Universal Robots PolyScope program: vg_palatz_cards.urp

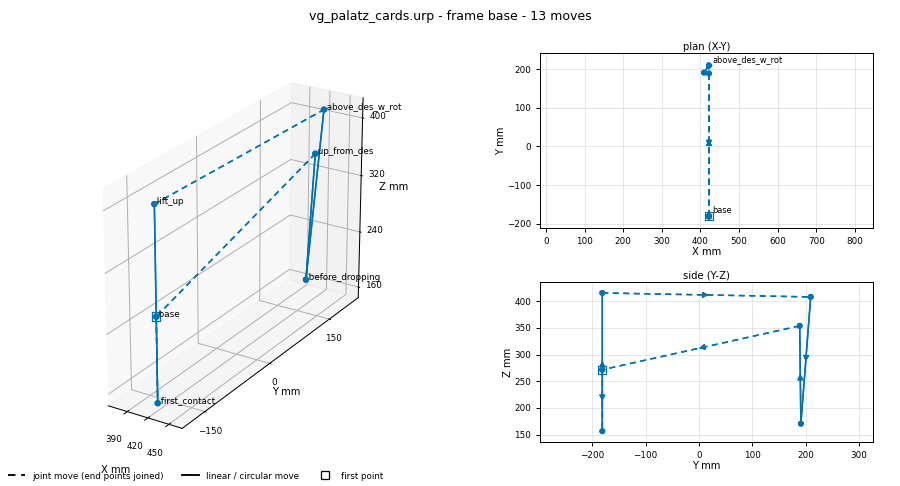
[picture p0: tool path of vg_palatz_cards.urp in frame base, 13 of 13 moves have a stored position in this frame; points joined in program order, loops and branches not executed]
Program vg_palatz_cards (installation=default directory=/programs/v_gripper_tm1326 createdIn=5.11.9.1010452 lastSavedIn=5.11.9.1010452 robotSerialNumber=20225200364)
Calibrated DH parameters: a=[0.00002, -0.569483, -0.54992, -0.00001, -0.000036, 0]; d=[0.180894, -146.691669, 192.918669, -46.053088, 0.119778, 0.115602]; alpha=[1.571425, -0.001534, 0.003359, 1.568739, -1.571477, 0]; deltaTheta=[0, 0.376258, -0.101074, -0.275185, -0.000002, 0]
Robot Program (runOnlyOnce=false)
  MoveJ speed 60 deg/s, acceleration 80 deg/s^2 (useActiveTCP=true) feature=Base
    Waypoint base: TCP in base x=421.909 y=-180.993 z=271.627 mm, rx=2.2364 ry=-2.2063 rz=0 rad; joints [-0.977, -80.029, -144.027, -45.908, 90.179, -1.705] deg
  MoveJ speed 60 deg/s, acceleration 80 deg/s^2 (useActiveTCP=true) feature=Base
    Waypoint first_contact: TCP in base x=421.917 y=-180.997 z=156.56 mm, rx=2.2364 ry=-2.2063 rz=-0.0001 rad; joints [-0.995, -95.96, -149.103, -24.902, 90.113, -1.657] deg
    URCap VG Grip (OnRobot, OnRobot A/S) dataModel(vg.grip.target.vacuum=5000.0, Variable(key=on_return, variable(name=on_return)))
  MoveL speed 250 mm/s, acceleration 1200 mm/s^2 (useActiveTCP=true) feature=Base
    Waypoint lift_up: TCP in base x=421.921 y=-180.985 z=415.39 mm, rx=2.2364 ry=-2.2063 rz=0 rad; joints [-0.961, -68.742, -134.04, -67.181, 90.213, -1.769] deg
  MoveJ speed 60 deg/s, acceleration 80 deg/s^2 (useActiveTCP=true) feature=Base
    Waypoint above_des_w_rot: TCP in base x=421.909 y=209.133 z=407.92 mm, rx=0.0024 ry=-3.1415 rz=-0.0002 rad; joints [48.032, -70.642, -133.729, -65.587, 90.219, 137.92] deg
  MoveL speed 250 mm/s, acceleration 1200 mm/s^2 (useActiveTCP=true) feature=Base
    Waypoint before_dropping: TCP in base x=409.206 y=190.757 z=170.596 mm, rx=0.0024 ry=-3.1415 rz=-0.0001 rad; joints [47.614, -92.993, -149.455, -27.515, 90.131, 137.632] deg
    URCap VG Release (OnRobot, OnRobot A/S)
    Waypoint up_from_des: TCP in base x=421.883 y=188.558 z=353.756 mm, rx=0.0024 ry=-3.1415 rz=-0.0001 rad; joints [46.178, -72.92, -138.459, -58.581, 90.212, 136.093] deg
  MoveJ speed 60 deg/s, acceleration 80 deg/s^2 (useActiveTCP=true) feature=Base
    Waypoint base: TCP in base x=421.909 y=-180.993 z=271.627 mm, rx=2.2364 ry=-2.2063 rz=0 rad; joints [-0.977, -80.029, -144.027, -45.908, 90.179, -1.705] deg
  MoveJ speed 60 deg/s, acceleration 80 deg/s^2 (useActiveTCP=true) feature=Base
    Waypoint first_contact: TCP in base x=421.917 y=-180.997 z=156.56 mm, rx=2.2364 ry=-2.2063 rz=-0.0001 rad; joints [-0.995, -95.96, -149.103, -24.902, 90.113, -1.657] deg
    URCap VG Grip (OnRobot, OnRobot A/S) dataModel(vg.grip.target.vacuum=5000.0, Variable(key=on_return, variable=on_return))
  MoveL speed 250 mm/s, acceleration 1200 mm/s^2 (useActiveTCP=true) feature=Base
    Waypoint lift_up: TCP in base x=421.921 y=-180.985 z=415.39 mm, rx=2.2364 ry=-2.2063 rz=0 rad; joints [-0.961, -68.742, -134.04, -67.181, 90.213, -1.769] deg
  MoveJ speed 60 deg/s, acceleration 80 deg/s^2 (useActiveTCP=true) feature=Base
    Waypoint above_des_w_rot: TCP in base x=421.909 y=209.133 z=407.92 mm, rx=0.0024 ry=-3.1415 rz=-0.0002 rad; joints [48.032, -70.642, -133.729, -65.587, 90.219, 137.92] deg
  MoveL speed 250 mm/s, acceleration 1200 mm/s^2 (useActiveTCP=true) feature=Base
    Waypoint before_dropping: TCP in base x=409.206 y=190.757 z=170.596 mm, rx=0.0024 ry=-3.1415 rz=-0.0001 rad; joints [47.614, -92.993, -149.455, -27.515, 90.131, 137.632] deg
    URCap VG Release (OnRobot, OnRobot A/S)
    Waypoint up_from_des: TCP in base x=421.883 y=188.558 z=353.756 mm, rx=0.0024 ry=-3.1415 rz=-0.0001 rad; joints [46.178, -72.92, -138.459, -58.581, 90.212, 136.093] deg
  MoveJ speed 60 deg/s, acceleration 80 deg/s^2 (useActiveTCP=true) feature=Base
    Waypoint base: TCP in base x=421.909 y=-180.993 z=271.627 mm, rx=2.2364 ry=-2.2063 rz=0 rad; joints [-0.977, -80.029, -144.027, -45.908, 90.179, -1.705] deg
    Halt
